// TIA Portal V18 export
TYPE "UDT_HSsAI"
// stored: IsFailsafeCompliant false
   STRUCT
      rHSBoilerRoomTemp : Real;   // 10.10 Температура в котельный
      rHSWaterPressure : Real;   // 10.09 Тиск в системы опалення
      rHSSupplyMainfoldTemp : Real;
      rOutdoorTemp_PLC_AI : Real;
   END_STRUCT;
END_TYPE
